(* CoDeSys 2.3 export: INVERNADEROS.EXP *)

(* POU Automatico/Invernaderos/Invernaderos, LD *)
PROGRAM Invernaderos
VAR
	(*Invernadero 1*)
	Cuenta1_1:BOOL; (*Planta 1 - Invernadero 1*)
	Cuenta2_1:BOOL; (*Planta 2 - Invernadero 1*)

	Final2_1:BOOL;
	Final1_1:BOOL;

	Invernadero1:Invernadero;
	Invernadero2: Invernadero;


	Cont1_1:CTU;
	Cont2_1:CTU;


	(*Invernadero 2*)
	Cuenta1_2:BOOL; (*Planta 1 - Invernadero 2*)
	Cuenta2_2:BOOL; (*Planta 2 - Invernadero 2*)

	Final1_2:BOOL;
	Final2_2:BOOL;

	Cont1_2:CTU;
	Cont2_2:CTU;


END_VAR
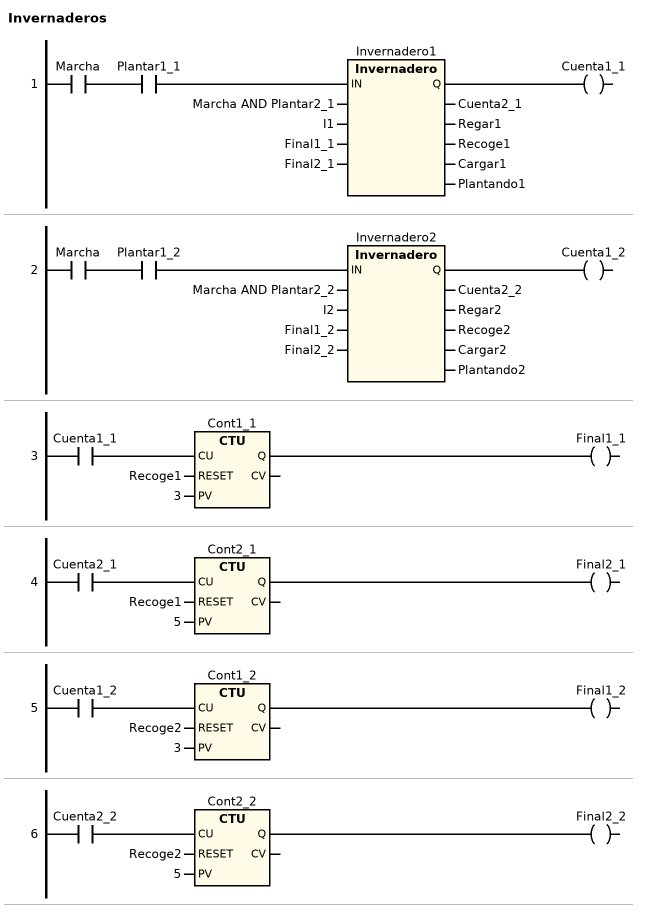
_LD_ (* Ladder Diagram *)
NETWORK 1
	[Marcha] - [Plantar1_1] - Invernadero1:Invernadero(*, Marcha AND Plantar2_1, I1, Final1_1, Final2_1, out 2 => Cuenta2_1, out 3 => Regar1, out 4 => Recoge1, out 5 => Cargar1, out 6 => Plantando1) --- (Cuenta1_1)
NETWORK 2
	[Marcha] - [Plantar1_2] - Invernadero2:Invernadero(*, Marcha AND Plantar2_2, I2, Final1_2, Final2_2, out 2 => Cuenta2_2, out 3 => Regar2, out 4 => Recoge2, out 5 => Cargar2, out 6 => Plantando2) --- (Cuenta1_2)
NETWORK 3
	[Cuenta1_1] - Cont1_1:CTU(CU: *, RESET: Recoge1, PV: 3) --- (Final1_1)
NETWORK 4
	[Cuenta2_1] - Cont2_1:CTU(CU: *, RESET: Recoge1, PV: 5) --- (Final2_1)
NETWORK 5
	[Cuenta1_2] - Cont1_2:CTU(CU: *, RESET: Recoge2, PV: 3) --- (Final1_2)
NETWORK 6
	[Cuenta2_2] - Cont2_2:CTU(CU: *, RESET: Recoge2, PV: 5) --- (Final2_2)
_END_LD_
(* the same logic as Structured Text *)
(* Network 1: see the listing above *)
(* Network 2: see the listing above *)
(* Network 3 *)
Cont1_1(CU := Cuenta1_1, RESET := Recoge1, PV := 3);
Final1_1 := Cont1_1.Q;
(* Network 4 *)
Cont2_1(CU := Cuenta2_1, RESET := Recoge1, PV := 5);
Final2_1 := Cont2_1.Q;
(* Network 5 *)
Cont1_2(CU := Cuenta1_2, RESET := Recoge2, PV := 3);
Final1_2 := Cont1_2.Q;
(* Network 6 *)
Cont2_2(CU := Cuenta2_2, RESET := Recoge2, PV := 5);
Final2_2 := Cont2_2.Q;
END_PROGRAM
